TYPE SystemStatusWord :
STRUCT
	// Das SystemStatusWord ist für die Interaktion zwischen den Reaktoren 	

	// Reaktor 1
	R1_Ready		:BOOL;
	R1_Activ		:BOOL;
	// Reaktor 2
	R2_Ready		:BOOL;
	R2_Activ		:BOOL;
	// Reaktor 3
	R3_Ready		:BOOL;
	R3_Activ		:BOOL;
	// Reaktor 4
	R4_Ready		:BOOL;
	R4_Activ		:BOOL;
	// Reaktor 5
	R5_Ready		:BOOL;
	R5_Activ		:BOOL;
	// Reaktor 6
	R6_Ready		:BOOL;
	R6_Activ		:BOOL;
	// Reaktor 7
	R7_Ready		:BOOL;
	R7_Activ		:BOOL;
END_STRUCT	
END_TYPE

(* stored: Version 1.1.0.1, ProductVersion 3.1.4024.12
   DUT SystemStatusWord: Id {eb27a699-e9d0-43a3-b599-3c1a56901629} *)
